Staubli VAL3: onF7Event.pgx

program onF7Event(bool& x_bSave[])
  local string l_sNew
  local bool l_bUndo
begin
   // look if the bButton is enable
  if bButton[6]
    //
    //  insert a new entry, it's use a FIFO politic
    //
    call alreadyExist(l_sNew,l_bUndo)
    if !l_bUndo and l_sNew!=""
      call axis:new(l_sNew,nIndex+1)
      nSelected=nIndex+1
      call buildList()
      call refreshStatic()
      // save it
      x_bSave=true
    endIf
  endIf
end
